KUKA KRL program: ENABLE_POSITION.src

&ACCESS RVO
&REL 2
DEFFCT BOOL ENABLE_POSITION( )

$STIFFNESS.STRATEGY = 10
$STIFFNESS.COMMIT = TRUE

RETURN TRUE

ENDFCT
